(* CoDeSys 2.3.9.41 project: VOS_Vorkuta_ASU_2_osmos_1.pro *)
(* Libraries: PID_Regulators.lib 6.11.19 15:29:27, Util.lib 18.5.10 15:14:28, STANDARD.LIB 4.10.05 11:14:46, IECSFC.LIB 13.4.06 15:51:28, GermesLib_1_4.lib 25.4.21 16:11:00, SYSLIBTIME.LIB 6.11.19 15:29:28, ANALYZATION.LIB 5.10.99 09:05:06 *)

(* PLC configuration (modules and I/O channels)
Fast discrete inputs [I_SIMPLE_INPUT] node 0, in %IB0 out %QB0 {ChannellName = Fast discrete inputs; Filtrationtime = 10000}
  DD1_DI_1 AT %IX0.0 [BitInput] Авария насоса Р03.01/01 {ChannellName = Enter name}
  DD1_DI_2 AT %IX0.1 [BitInput] Авария насоса Р03.01/02 {ChannellName = Enter name}
  DD1_DI_3 AT %IX0.2 [BitInput] эк.манометр PIS03.01/01 после насоса Р03.01/01 {ChannellName = Enter name}
  DD1_DI_4 AT %IX0.3 [BitInput] эк.манометр PIS03.01/02 после насоса Р03.01/02 {ChannellName = Enter name}
Discrete inputs [ID130] node 1, in %IB1 out %QB1 {ChannellName = Discrete inputs; Filtrationtime_GeneralINP = 10; PinCount = 12; Visibility = No}
  AT %IB1.0 [ByteInput] 8 discrete inputs {ChannellName = Enter name}
  AT %IB1.1 [ByteInput] 4 discrete inputs {ChannellName = Enter name}
Fast discrete outputs [OWEN_ID570] node 2, in %IB2 out %QB2 {ChannellName = Fast discrete outputs; SafeValueBool = FALSE; SafeValueBool = FALSE; SafeValueBool = FALSE; SafeValueBool = FALSE; Visibility = No}
  DD1_DO_1 AT %QX2.0 [BitOutput] Fast discrete output 1 {ChannellName = Enter name}
  DD1_DO_2 AT %QX2.1 [BitOutput] Fast discrete output 2 {ChannellName = Enter name}
  DD1_DO_3 AT %QX2.2 [BitOutput] Fast discrete output 3 {ChannellName = Enter name}
  DD1_DO_4 AT %QX2.3 [BitOutput] Fast discrete output 4 {ChannellName = Enter name}
Discrete outputs [ID131] node 3, in %IB3 out %QB3 {ChannellName = Discrete outputs; SafeValueByte = 0; Visibility = No}
  AT %QB3.0 [ByteOutput] 8 discrete outputs {ChannellName = Enter name}
  AT %QB3.1 [ByteOutput] 8 discrete outputs {ChannellName = Enter name}
Fast analog inputs [ID125] node 4, in %IB4 out %QB4 {ChannellName = Fast analog inputs; Flt_Comm = 50Hz 2Por}
  DD1_AI_1 AT %IR4.0 [FloatInputP] LT02.03 уровень в емкости V02.07 {ChannellName = Fast analog input; AIN_TYPE = 0-20 mA; Peak_Filtr = 200; Flt_Ch = Off; TauRC = 10; MinFV = 0; MaxFV = 20}
  DD1_AI_2 AT %IR4.1 [FloatInputP] датчик давления РТ03.01/01 {ChannellName = Fast analog input; AIN_TYPE = 0-20 mA; Peak_Filtr = 200; Flt_Ch = Off; TauRC = 10; MinFV = 0; MaxFV = 20}
  DD1_AI_3 AT %IR4.2 [FloatInputP] датчик давления РТ03.02/01 {ChannellName = Fast analog input; AIN_TYPE = 0-20 mA; Peak_Filtr = 200; Flt_Ch = Off; TauRC = 10; MinFV = 0; MaxFV = 20}
  DD1_AI_4 AT %IR4.3 [FloatInputP] датчик давления РТ03.03/01 {ChannellName = Fast analog input; AIN_TYPE = 0-20 mA; Peak_Filtr = 200; Flt_Ch = Off; TauRC = 10; MinFV = 0; MaxFV = 20}
  DD1_AI_5 AT %IR4.4 [FloatInputP] датчик давления РТ03.04/01 {ChannellName = Fast analog input; AIN_TYPE = 0-20 mA; Peak_Filtr = 200; Flt_Ch = Off; TauRC = 10; MinFV = 0; MaxFV = 20}
  DD1_AI_6 AT %IR4.5 [FloatInputP] кондуктомер QIT03.01/01 осн.осмос {ChannellName = Fast analog input; AIN_TYPE = 0-20 mA; Peak_Filtr = 200; Flt_Ch = Off; TauRC = 10; MinFV = 0; MaxFV = 20}
  DD1_AI_7 AT %IR4.6 [FloatInputP] расходомер FIT03.02/01 осн.осмос {ChannellName = Fast analog input; AIN_TYPE = 0-20 mA; Peak_Filtr = 200; Flt_Ch = Off; TauRC = 10; MinFV = 0; MaxFV = 20}
  DD1_AI_8 AT %IR4.7 [FloatInputP] расходомер FIT03.03/01 осн.осмос {ChannellName = Fast analog input; AIN_TYPE = 0-20 mA; Peak_Filtr = 200; Flt_Ch = Off; TauRC = 10; MinFV = 0; MaxFV = 20}
  AT %IW4.8 [WordInput] AI read time (10ms) {ChannellName = Enter name}
Analog outputs [ID126] node 5, in %IB5 out %QB5 {ChannellName = Analog outputs}
  DD1_AO_1 AT %QR5.0 [FloatOutputP] производительность осн.доз.насоса Р03.02/01 {ChannellName = Analog output; AOUT_TYPE = 4-20 mA; SafeValueREAL = 0.0}
  DD1_AO_2 AT %QR5.1 [FloatOutputP] производительность рез.доз.насоса Р03.02/02 {ChannellName = Analog output; AOUT_TYPE = 4-20 mA; SafeValueREAL = 0.0}
  DD1_AO_3 AT %QR5.2 [FloatOutputP] резерв {ChannellName = Analog output; AOUT_TYPE = 4-20 mA; SafeValueREAL = 0.0}
  DD1_AO_4 AT %QR5.3 [FloatOutputP] резерв {ChannellName = Analog output; AOUT_TYPE = 4-20 mA; SafeValueREAL = 0.0}
Special input [ID103] node 6, in %IB6 out %QB6 {ChannellName = Special input}
  AT %IX6.0 [BitInput] Special input {ChannellName = Enter name}
Special output [ID104] node 7, in %IB7 out %QB7 {ChannellName = Special output}
  AT %QX7.0 [BitOutput] Special output {ChannellName = Enter name}
ModBus (Master) [MODBUS_MASTER_ID450] node 8, in %IB8 out %QB8 {ChannellName = ModBus (Master); Visibility = No}
  AT %QD8.0 [DWordOutput] Last address {ChannellName = Enter name}
  AT %QW8.1 [WordOutput] Last error {ChannellName = Enter name}
  RS-485-1 [COM1_USART] node 0, in %IB8.0 out %QB8.0 {ChannellName = RS-485-1; CommunicationSpeed = 9600; Parity = NO PARITY CHECK; BitLength = 8 bits; StopLength = One stop bit; InterfaceType = RS485; FrameOriented = RTU; Timeout = 5; Visibility = No}
  Universal Modbus device [ID2000] node 1, in %IB8.1 out %QB8.1 {ChannellName = Universal Modbus device; ModuleIP = 10:0:0:223; ServiceTimeout = 150; TCPport = 502; NetMode = Serial; ModuleSlaveAddress = 11; RequestType = By poll time; PeriodOfService = 100; Visibility = No; RepeatCounter = 0; ByteSequence = Native}
    AT %QB8.1.0 [ComChannel] Command (0xff - Start) {ChannellName = Enter name}
    Real input module [ID2007] node 0, in %IB8.1.0 out %QB8.1.0 {ChannellName = float input module; ModbusAddress = 512; Command_read_regs = Read holding Registers  (0x03); Visibility = No}
      PT030102rawValue AT %QD8.1.0.0 [FloatOutput] {ChannellName = Enter name}
    Real input module [ID2007] node 1, in %IB8.1.1 out %QB8.1.1 {ChannellName = float input module; ModbusAddress = 514; Command_read_regs = Read holding Registers  (0x03); Visibility = No}
      PT030202rawValue AT %QD8.1.1.0 [FloatOutput] {ChannellName = Enter name}
    Real input module [ID2007] node 2, in %IB8.1.2 out %QB8.1.2 {ChannellName = float input module; ModbusAddress = 516; Command_read_regs = Read holding Registers  (0x03); Visibility = No}
      PT030302rawValue AT %QD8.1.2.0 [FloatOutput] {ChannellName = Enter name}
    Real input module [ID2007] node 3, in %IB8.1.3 out %QB8.1.3 {ChannellName = float input module; ModbusAddress = 518; Command_read_regs = Read holding Registers  (0x03); Visibility = No}
      PT030402rawValue AT %QD8.1.3.0 [FloatOutput] {ChannellName = Enter name}
    Real input module [ID2007] node 4, in %IB8.1.4 out %QB8.1.4 {ChannellName = float input module; ModbusAddress = 520; Command_read_regs = Read holding Registers  (0x03); Visibility = No}
      QIT030102rawValue AT %QD8.1.4.0 [FloatOutput] {ChannellName = Enter name}
    Real input module [ID2007] node 5, in %IB8.1.5 out %QB8.1.5 {ChannellName = float input module; ModbusAddress = 522; Command_read_regs = Read holding Registers  (0x03); Visibility = No}
      FIT030202rawValue AT %QD8.1.5.0 [FloatOutput] {ChannellName = Enter name}
    Real input module [ID2007] node 6, in %IB8.1.6 out %QB8.1.6 {ChannellName = float input module; ModbusAddress = 524; Command_read_regs = Read holding Registers  (0x03); Visibility = No}
      FIT030302rawValue AT %QD8.1.6.0 [FloatOutput] {ChannellName = Enter name}
      reserve_FIT030101rawValue AT %QD8.1.7.0 [FloatOutput] {ChannellName = Enter name}
    Register input module [ID2003] node 8, in %IB8.1.8 out %QB8.1.8 {ChannellName = Register input module; ModbusAddress = 529; Command_read_regs = Read input registers  (0x04); Visibility = No}
      DI_bit_mask_DD2 AT %QW8.1.8.0 [WordOutput] {ChannellName = Enter name}
    Register input module [ID2003] node 9, in %IB8.1.9 out %QB8.1.9 {ChannellName = Register input module; ModbusAddress = 532; Command_read_regs = Read input registers  (0x04); Visibility = No}
      stat_word_P030601_PLC AT %QW8.1.9.0 [WordOutput] {ChannellName = Enter name}
    Register input module [ID2003] node 10, in %IB8.1.10 out %QB8.1.10 {ChannellName = Register input module; ModbusAddress = 535; Command_read_regs = Read input registers  (0x04); Visibility = No}
      stat_word_P030602_PLC AT %QW8.1.10.0 [WordOutput] {ChannellName = Enter name}
  Universal Modbus device [ID2000] node 2, in %IB8.2 out %QB8.2 {ChannellName = Universal Modbus device; ModuleIP = 10:0:0:223; ServiceTimeout = 150; TCPport = 502; NetMode = Serial; ModuleSlaveAddress = 1; RequestType = By value change; PeriodOfService = 100; Visibility = No; RepeatCounter = 0; ByteSequence = Native}
    AT %QB8.2.0 [ComChannel] Command (0xff - Start) {ChannellName = Enter name}
    Register output module [ID2004] node 0, in %IB8.2.0 out %QB8.2.0 {ChannellName = Register; ModbusAddress = 528; Command_write_one_reg = Write multiple registers(0x10); Visibility = No}
      DO_bit_mask_DD2 AT %QW8.2.0.0 [WordOutput] {ChannellName = Enter name}
    Register output module [ID2004] node 1, in %IB8.2.1 out %QB8.2.1 {ChannellName = Register; ModbusAddress = 530; Command_write_one_reg = Write multiple registers(0x10); Visibility = No}
      com_word_P030601_PLC AT %QW8.2.1.0 [WordOutput] {ChannellName = Enter name}
    Register output module [ID2004] node 2, in %IB8.2.2 out %QB8.2.2 {ChannellName = Register; ModbusAddress = 531; Command_write_one_reg = Write multiple registers(0x10); Visibility = No}
      set_freq_P030601_PLC AT %QW8.2.2.0 [WordOutput] {ChannellName = Enter name}
    Register output module [ID2004] node 3, in %IB8.2.3 out %QB8.2.3 {ChannellName = Register; ModbusAddress = 533; Command_write_one_reg = Write multiple registers(0x10); Visibility = No}
      com_word_P030602_PLC AT %QW8.2.3.0 [WordOutput] {ChannellName = Enter name}
    Register output module [ID2004] node 4, in %IB8.2.4 out %QB8.2.4 {ChannellName = Register; ModbusAddress = 534; Command_write_one_reg = Write multiple registers(0x10); Visibility = No}
      set_freq_P030602_PLC AT %QW8.2.4.0 [WordOutput] {ChannellName = Enter name}
ModBus (Master) [MODBUS_MASTER_ID450] node 9, in %IB9 out %QB9 {ChannellName = ModBus (Master); Visibility = No}
  AT %QD9.0 [DWordOutput] Last address {ChannellName = Enter name}
  AT %QW9.1 [WordOutput] Last error {ChannellName = Enter name}
  RS-232 [COM2_USART] node 0, in %IB9.0 out %QB9.0 {ChannellName = RS-232; CommunicationSpeed = 115200; Parity = NO PARITY CHECK; BitLength = 8 bits; StopLength = One stop bit; InterfaceType = RS232; FrameOriented = RTU; Timeout = 5; Visibility = No}
  Universal Modbus device [ID2000] node 1, in %IB9.1 out %QB9.1 {ChannellName = Universal Modbus device; ModuleIP = 10:0:0:223; ServiceTimeout = 150; TCPport = 502; NetMode = Serial; ModuleSlaveAddress = 1; RequestType = By poll time; PeriodOfService = 50; Visibility = No; RepeatCounter = 0; ByteSequence = Native}
    AT %QB9.1.0 [ComChannel] Command (0xff - Start) {ChannellName = Enter name}
PANsetWordP0302 AT %QW9.1.0.0 [WordOutput] {ChannellName = Enter name}
PAN_LT0203maxValue AT %QD9.1.1.0 [FloatOutput] {ChannellName = Enter name}
PANsetMaxPumpDosingValueP0302 AT %QD9.1.2.0 [FloatOutput] {ChannellName = Enter name}
PANsetKoeffPropotrionalityP0302 AT %QD9.1.3.0 [FloatOutput] {ChannellName = Enter name}
PAN_CHECKING_DELAY_TIME AT %QW9.1.4.0 [WordOutput] {ChannellName = Enter name}
PAN_DELAY_REPEATED_START_SEC AT %QW9.1.5.0 [WordOutput] {ChannellName = Enter name}
PAN_DELAY_TO_OFF_VALVE AT %QW9.1.6.0 [WordOutput] {ChannellName = Enter name}
PAN_DELAY_TO_CHECK_PT0301 AT %QW9.1.7.0 [WordOutput] {ChannellName = Enter name}
PAN_DELAY_TO_SWITCH_VALVE AT %QW9.1.8.0 [WordOutput] {ChannellName = Enter name}
PAN_DELAY_TO_CLOSE_VALVE AT %QW9.1.9.0 [WordOutput] {ChannellName = Enter name}
PAN_FIT030201maxValue AT %QD9.1.10.0 [FloatOutput] {ChannellName = Enter name}
PAN_FIT030301maxValue AT %QD9.1.11.0 [FloatOutput] {ChannellName = Enter name}
PAN_FIT030202maxValue AT %QD9.1.12.0 [FloatOutput] {ChannellName = Enter name}
PAN_FIT030302maxValue AT %QD9.1.13.0 [FloatOutput] {ChannellName = Enter name}
PAN_QIT030101maxValue AT %QD9.1.14.0 [FloatOutput] {ChannellName = Enter name}
PAN_QIT030102maxValue AT %QD9.1.15.0 [FloatOutput] {ChannellName = Enter name}
PAN_PT030101maxValue AT %QD9.1.16.0 [FloatOutput] {ChannellName = Enter name}
PAN_PT030201maxValue AT %QD9.1.17.0 [FloatOutput] {ChannellName = Enter name}
PAN_PT030301maxValue AT %QD9.1.18.0 [FloatOutput] {ChannellName = Enter name}
PAN_PT030401maxValue AT %QD9.1.19.0 [FloatOutput] {ChannellName = Enter name}
PAN_PT030102maxValue AT %QD9.1.20.0 [FloatOutput] {ChannellName = Enter name}
PAN_PT030202maxValue AT %QD9.1.21.0 [FloatOutput] {ChannellName = Enter name}
PAN_PT030302maxValue AT %QD9.1.22.0 [FloatOutput] {ChannellName = Enter name}
PAN_PT030402maxValue AT %QD9.1.23.0 [FloatOutput] {ChannellName = Enter name}
PANsetWordOsmos AT %QW9.1.24.0 [WordOutput] {ChannellName = Enter name}
PAN_PT0301startValue AT %QD9.1.25.0 [FloatOutput] {ChannellName = Enter name}
PAN_FIT0303setValue AT %QD9.1.26.0 [FloatOutput] {ChannellName = Enter name}
PAN_PT0302setMaxValue AT %QD9.1.27.0 [FloatOutput] {ChannellName = Enter name}
PAN_PT0303setMaxValue AT %QD9.1.28.0 [FloatOutput] {ChannellName = Enter name}
PAN_PT0304setMaxValue AT %QD9.1.29.0 [FloatOutput] {ChannellName = Enter name}
PAN_KP_F_P030601 AT %QD9.1.30.0 [FloatOutput] {ChannellName = Enter name}
PAN_I_F_P030601 AT %QD9.1.31.0 [FloatOutput] {ChannellName = Enter name}
%MPAN_D_F_P030601 AT %QD9.1.32.0 [FloatOutput] {ChannellName = Enter name}
%MPAN_KP_P_P030601 AT %QD9.1.33.0 [FloatOutput] {ChannellName = Enter name}
PAN_I_P_P030601 AT %QD9.1.34.0 [FloatOutput] {ChannellName = Enter name}
PAN_D_P_P030601 AT %QD9.1.35.0 [FloatOutput] {ChannellName = Enter name}
PAN_KP_F_P030602 AT %QD9.1.36.0 [FloatOutput] {ChannellName = Enter name}
PAN_I_F_P030602 AT %QD9.1.37.0 [FloatOutput] {ChannellName = Enter name}
PAN_D_F_P030602 AT %QD9.1.38.0 [FloatOutput] {ChannellName = Enter name}
PAN_KP_P_P030602 AT %QD9.1.39.0 [FloatOutput] {ChannellName = Enter name}
PAN_I_P_P030602 AT %QD9.1.40.0 [FloatOutput] {ChannellName = Enter name}
PAN_D_P_P030602 AT %QD9.1.41.0 [FloatOutput] {ChannellName = Enter name}
PAN_FIT0303_SetCascade AT %QD9.1.42.0 [FloatOutput] {ChannellName = Enter name}
ID2003NoNoINTRegister input module+ AT %QW9.1.43.0 [WordOutput] B	+%QB	+%MB	+%MPAN_valuesActivator {ChannellName = Enter name}
PAN_V0207maxHeight AT %QD9.1.44.0 [FloatOutput] {ChannellName = Enter name}
PAN_V0207minHeight AT %QD9.1.45.0 [FloatOutput] {ChannellName = Enter name}
Universal Modbus device [ID2000] node 2, in %IB9.2 out %QB9.2 {ChannellName = Universal Modbus device; ModuleIP = 10:0:0:223; ServiceTimeout = 150; TCPport = 502; NetMode = Serial; ModuleSlaveAddress = 1; RequestType = Both; PeriodOfService = 100; Visibility = No; RepeatCounter = 0; ByteSequence = Native}
  AT %QB9.2.0 [ComChannel] Command (0xff - Start) {ChannellName = Enter name}
  Register output module [ID2004] node 0, in %IB9.2.0 out %QB9.2.0 {ChannellName = Register; ModbusAddress = 271; Command_write_one_reg = Write multiple registers(0x10); Visibility = No}
    PANstatWordP0302 AT %QW9.2.0.0 [WordOutput] {ChannellName = Enter name}
  Register output module [ID2004] node 1, in %IB9.2.1 out %QB9.2.1 {ChannellName = Register; ModbusAddress = 272; Command_write_one_reg = Write multiple registers(0x10); Visibility = No}
    PANdaysOfWorkP030201 AT %QW9.2.1.0 [WordOutput] {ChannellName = Enter name}
  Register output module [ID2004] node 2, in %IB9.2.2 out %QB9.2.2 {ChannellName = Register; ModbusAddress = 273; Command_write_one_reg = Write multiple registers(0x10); Visibility = No}
    PANhoursOfWorkP030201 AT %QW9.2.2.0 [WordOutput] {ChannellName = Enter name}
  Register output module [ID2004] node 3, in %IB9.2.3 out %QB9.2.3 {ChannellName = Register; ModbusAddress = 274; Command_write_one_reg = Write multiple registers(0x10); Visibility = No}
    PANminutesOfWorkP030201 AT %QW9.2.3.0 [WordOutput] {ChannellName = Enter name}
  Register output module [ID2004] node 4, in %IB9.2.4 out %QB9.2.4 {ChannellName = Register; ModbusAddress = 275; Command_write_one_reg = Write multiple registers(0x10); Visibility = No}
    PANsecondsOfWorkP030201 AT %QW9.2.4.0 [WordOutput] {ChannellName = Enter name}
  Register output module [ID2004] node 5, in %IB9.2.5 out %QB9.2.5 {ChannellName = Register; ModbusAddress = 276; Command_write_one_reg = Write multiple registers(0x10); Visibility = No}
    PANtoNextStartP030201timer AT %QW9.2.5.0 [WordOutput] {ChannellName = Enter name}
  Register output module [ID2004] node 6, in %IB9.2.6 out %QB9.2.6 {ChannellName = Register; ModbusAddress = 277; Command_write_one_reg = Write multiple registers(0x10); Visibility = No}
    PANdaysOfWorkP030202 AT %QW9.2.6.0 [WordOutput] {ChannellName = Enter name}
  Register output module [ID2004] node 7, in %IB9.2.7 out %QB9.2.7 {ChannellName = Register; ModbusAddress = 278; Command_write_one_reg = Write multiple registers(0x10); Visibility = No}
    PANhoursOfWorkP030202 AT %QW9.2.7.0 [WordOutput] {ChannellName = Enter name}
  Register output module [ID2004] node 8, in %IB9.2.8 out %QB9.2.8 {ChannellName = Register; ModbusAddress = 279; Command_write_one_reg = Write multiple registers(0x10); Visibility = No}
    PANminutesOfWorkP030202 AT %QW9.2.8.0 [WordOutput] {ChannellName = Enter name}
  Register output module [ID2004] node 9, in %IB9.2.9 out %QB9.2.9 {ChannellName = Register; ModbusAddress = 280; Command_write_one_reg = Write multiple registers(0x10); Visibility = No}
    PANsecondsOfWorkP030202 AT %QW9.2.9.0 [WordOutput] {ChannellName = Enter name}
  Register output module [ID2004] node 10, in %IB9.2.10 out %QB9.2.10 {ChannellName = Register; ModbusAddress = 281; Command_write_one_reg = Write multiple registers(0x10); Visibility = No}
    PANtoNextStartP030202timer AT %QW9.2.10.0 [WordOutput] {ChannellName = Enter name}
  Real output module [ID2008] node 11, in %IB9.2.11 out %QB9.2.11 {ChannellName = float output module; ModbusAddress = 282; Command_write_regs = Preset multiple Registers (0x10); Visibility = No}
    PANcounterP030201 AT %QD9.2.11.0 [FloatOutput] {ChannellName = Enter name}
  Real output module [ID2008] node 12, in %IB9.2.12 out %QB9.2.12 {ChannellName = float output module; ModbusAddress = 284; Command_write_regs = Preset multiple Registers (0x10); Visibility = No}
    PANcounterP030202 AT %QD9.2.12.0 [FloatOutput] {ChannellName = Enter name}
  Real output module [ID2008] node 13, in %IB9.2.13 out %QB9.2.13 {ChannellName = float output module; ModbusAddress = 286; Command_write_regs = Preset multiple Registers (0x10); Visibility = No}
    PAN_FIT0301realValue AT %QD9.2.13.0 [FloatOutput] {ChannellName = Enter name}
  Real output module [ID2008] node 14, in %IB9.2.14 out %QB9.2.14 {ChannellName = float output module; ModbusAddress = 288; Command_write_regs = Preset multiple Registers (0x10); Visibility = No}
    PAN_PT030101realValue AT %QD9.2.14.0 [FloatOutput] {ChannellName = Enter name}
  Real output module [ID2008] node 15, in %IB9.2.15 out %QB9.2.15 {ChannellName = float output module; ModbusAddress = 290; Command_write_regs = Preset multiple Registers (0x10); Visibility = No}
    PAN_PT030201realValue AT %QD9.2.15.0 [FloatOutput] {ChannellName = Enter name}
  Real output module [ID2008] node 16, in %IB9.2.16 out %QB9.2.16 {ChannellName = float output module; ModbusAddress = 292; Command_write_regs = Preset multiple Registers (0x10); Visibility = No}
    PAN_PT030301realValue AT %QD9.2.16.0 [FloatOutput] {ChannellName = Enter name}
  Real output module [ID2008] node 17, in %IB9.2.17 out %QB9.2.17 {ChannellName = float output module; ModbusAddress = 294; Command_write_regs = Preset multiple Registers (0x10); Visibility = No}
    PAN_FIT030301realValue AT %QD9.2.17.0 [FloatOutput] {ChannellName = Enter name}
  Real output module [ID2008] node 18, in %IB9.2.18 out %QB9.2.18 {ChannellName = float output module; ModbusAddress = 296; Command_write_regs = Preset multiple Registers (0x10); Visibility = No}
    PAN_PT030102realValue AT %QD9.2.18.0 [FloatOutput] {ChannellName = Enter name}
  Real output module [ID2008] node 19, in %IB9.2.19 out %QB9.2.19 {ChannellName = float output module; ModbusAddress = 298; Command_write_regs = Preset multiple Registers (0x10); Visibility = No}
    PAN_PT030202realValue AT %QD9.2.19.0 [FloatOutput] {ChannellName = Enter name}
  Real output module [ID2008] node 20, in %IB9.2.20 out %QB9.2.20 {ChannellName = float output module; ModbusAddress = 300; Command_write_regs = Preset multiple Registers (0x10); Visibility = No}
    PAN_PT030302realValue AT %QD9.2.20.0 [FloatOutput] {ChannellName = Enter name}
  Real output module [ID2008] node 21, in %IB9.2.21 out %QB9.2.21 {ChannellName = float output module; ModbusAddress = 302; Command_write_regs = Preset multiple Registers (0x10); Visibility = No}
    PAN_FIT030302realValue AT %QD9.2.21.0 [FloatOutput] {ChannellName = Enter name}
  Real output module [ID2008] node 22, in %IB9.2.22 out %QB9.2.22 {ChannellName = float output module; ModbusAddress = 304; Command_write_regs = Preset multiple Registers (0x10); Visibility = No}
    PAN_PT030401realValue AT %QD9.2.22.0 [FloatOutput] {ChannellName = Enter name}
  Real output module [ID2008] node 23, in %IB9.2.23 out %QB9.2.23 {ChannellName = float output module; ModbusAddress = 306; Command_write_regs = Preset multiple Registers (0x10); Visibility = No}
    PAN_FIT030201realValue AT %QD9.2.23.0 [FloatOutput] {ChannellName = Enter name}
  Real output module [ID2008] node 24, in %IB9.2.24 out %QB9.2.24 {ChannellName = float output module; ModbusAddress = 308; Command_write_regs = Preset multiple Registers (0x10); Visibility = No}
    PAN_QIT030101realValue AT %QD9.2.24.0 [FloatOutput] {ChannellName = Enter name}
  Real output module [ID2008] node 25, in %IB9.2.25 out %QB9.2.25 {ChannellName = float output module; ModbusAddress = 310; Command_write_regs = Preset multiple Registers (0x10); Visibility = No}
    PAN_PT030402realValue AT %QD9.2.25.0 [FloatOutput] {ChannellName = Enter name}
  Real output module [ID2008] node 26, in %IB9.2.26 out %QB9.2.26 {ChannellName = float output module; ModbusAddress = 312; Command_write_regs = Preset multiple Registers (0x10); Visibility = No}
    PAN_FIT030202realValue AT %QD9.2.26.0 [FloatOutput] {ChannellName = Enter name}
  Real output module [ID2008] node 27, in %IB9.2.27 out %QB9.2.27 {ChannellName = float output module; ModbusAddress = 314; Command_write_regs = Preset multiple Registers (0x10); Visibility = No}
    PAN_QIT030102realValue AT %QD9.2.27.0 [FloatOutput] {ChannellName = Enter name}
  Register output module [ID2004] node 28, in %IB9.2.28 out %QB9.2.28 {ChannellName = Register; ModbusAddress = 316; Command_write_one_reg = Write multiple registers(0x10); Visibility = No}
    PANstatWordOsmos AT %QW9.2.28.0 [WordOutput] {ChannellName = Enter name}
  Register output module [ID2004] node 29, in %IB9.2.29 out %QB9.2.29 {ChannellName = Register; ModbusAddress = 317; Command_write_one_reg = Write multiple registers(0x10); Visibility = No}
    PANdaysOfWorkOsmos1 AT %QW9.2.29.0 [WordOutput] {ChannellName = Enter name}
  Register output module [ID2004] node 30, in %IB9.2.30 out %QB9.2.30 {ChannellName = Register; ModbusAddress = 318; Command_write_one_reg = Write multiple registers(0x10); Visibility = No}
    PANhoursOfWorkOsmos1 AT %QW9.2.30.0 [WordOutput] {ChannellName = Enter name}
  Register output module [ID2004] node 31, in %IB9.2.31 out %QB9.2.31 {ChannellName = Register; ModbusAddress = 319; Command_write_one_reg = Write multiple registers(0x10); Visibility = No}
    PANminutesOfWorkOsmos1 AT %QW9.2.31.0 [WordOutput] {ChannellName = Enter name}
  Register output module [ID2004] node 32, in %IB9.2.32 out %QB9.2.32 {ChannellName = Register; ModbusAddress = 320; Command_write_one_reg = Write multiple registers(0x10); Visibility = No}
    PANsecondsOfWorkOsmos1 AT %QW9.2.32.0 [WordOutput] {ChannellName = Enter name}
  Register output module [ID2004] node 33, in %IB9.2.33 out %QB9.2.33 {ChannellName = Register; ModbusAddress = 321; Command_write_one_reg = Write multiple registers(0x10); Visibility = No}
    PANtoNextStartOsmos1timer AT %QW9.2.33.0 [WordOutput] {ChannellName = Enter name}
  Real output module [ID2008] node 34, in %IB9.2.34 out %QB9.2.34 {ChannellName = float output module; ModbusAddress = 322; Command_write_regs = Preset multiple Registers (0x10); Visibility = No}
    PANcounterOsmos1 AT %QD9.2.34.0 [FloatOutput] {ChannellName = Enter name}
  Real output module [ID2008] node 35, in %IB9.2.35 out %QB9.2.35 {ChannellName = float output module; ModbusAddress = 324; Command_write_regs = Preset multiple Registers (0x10); Visibility = No}
    PANcounterOsmos2 AT %QD9.2.35.0 [FloatOutput] {ChannellName = Enter name}
  Register output module [ID2004] node 36, in %IB9.2.36 out %QB9.2.36 {ChannellName = Register; ModbusAddress = 326; Command_write_one_reg = Write multiple registers(0x10); Visibility = No}
    PANdaysOfWorkOsmos2 AT %QW9.2.36.0 [WordOutput] {ChannellName = Enter name}
  Register output module [ID2004] node 37, in %IB9.2.37 out %QB9.2.37 {ChannellName = Register; ModbusAddress = 327; Command_write_one_reg = Write multiple registers(0x10); Visibility = No}
    PANhoursOfWorkOsmos2 AT %QW9.2.37.0 [WordOutput] {ChannellName = Enter name}
  Register output module [ID2004] node 38, in %IB9.2.38 out %QB9.2.38 {ChannellName = Register; ModbusAddress = 328; Command_write_one_reg = Write multiple registers(0x10); Visibility = No}
    PANminutesOfWorkOsmos2 AT %QW9.2.38.0 [WordOutput] {ChannellName = Enter name}
  Register output module [ID2004] node 39, in %IB9.2.39 out %QB9.2.39 {ChannellName = Register; ModbusAddress = 329; Command_write_one_reg = Write multiple registers(0x10); Visibility = No}
    PANsecondsOfWorkOsmos2 AT %QW9.2.39.0 [WordOutput] {ChannellName = Enter name}
  Register output module [ID2004] node 40, in %IB9.2.40 out %QB9.2.40 {ChannellName = Register; ModbusAddress = 330; Command_write_one_reg = Write multiple registers(0x10); Visibility = No}
    PANtoNextStartOsmos2timer AT %QW9.2.40.0 [WordOutput] {ChannellName = Enter name}
  Register output module [ID2004] node 41, in %IB9.2.41 out %QB9.2.41 {ChannellName = Register; ModbusAddress = 331; Command_write_one_reg = Write multiple registers(0x10); Visibility = No}
    PANmainViewBools AT %QW9.2.41.0 [WordOutput] {ChannellName = Enter name}
PAN_BMT_Flow AT %QD9.2.42.0 [FloatOutput] {ChannellName = Enter name}
32bit output module [ID2006] node 43, in %IB9.2.43 out %QB9.2.43 {ChannellName = 32 bit output module; ModbusAddress = 336; Command_write_regs = Preset multiple Registers (0x10); Visibility = No}
  PANalarms AT %QD9.2.43.0 [DWordOutput] {ChannellName = Enter name}
Real output module [ID2008] node 44, in %IB9.2.44 out %QB9.2.44 {ChannellName = float output module; ModbusAddress = 338; Command_write_regs = Preset multiple Registers (0x10); Visibility = No}
  PAN_currentValue_PT0301startValue AT %QD9.2.44.0 [FloatOutput] {ChannellName = Enter name}
Real output module [ID2008] node 45, in %IB9.2.45 out %QB9.2.45 {ChannellName = float output module; ModbusAddress = 340; Command_write_regs = Preset multiple Registers (0x10); Visibility = No}
  PAN_currentValue_FIT0303setValue AT %QD9.2.45.0 [FloatOutput] {ChannellName = Enter name}
Real output module [ID2008] node 46, in %IB9.2.46 out %QB9.2.46 {ChannellName = float output module; ModbusAddress = 342; Command_write_regs = Preset multiple Registers (0x10); Visibility = No}
  PAN_currentValue_PT0302setMaxValue AT %QD9.2.46.0 [FloatOutput] {ChannellName = Enter name}
Real output module [ID2008] node 47, in %IB9.2.47 out %QB9.2.47 {ChannellName = float output module; ModbusAddress = 344; Command_write_regs = Preset multiple Registers (0x10); Visibility = No}
  PAN_currentValue_PT0303setMaxValue AT %QD9.2.47.0 [FloatOutput] {ChannellName = Enter name}
Real output module [ID2008] node 48, in %IB9.2.48 out %QB9.2.48 {ChannellName = float output module; ModbusAddress = 346; Command_write_regs = Preset multiple Registers (0x10); Visibility = No}
  PAN_currentValue_PT0304setMaxValue AT %QD9.2.48.0 [FloatOutput] {ChannellName = Enter name}
Real output module [ID2008] node 49, in %IB9.2.49 out %QB9.2.49 {ChannellName = float output module; ModbusAddress = 348; Command_write_regs = Preset multiple Registers (0x10); Visibility = No}
  PAN_currentValue_FIT0303_SetCascade AT %QD9.2.49.0 [FloatOutput] {ChannellName = Enter name}
Real output module [ID2008] node 50, in %IB9.2.50 out %QB9.2.50 {ChannellName = float output module; ModbusAddress = 350; Command_write_regs = Preset multiple Registers (0x10); Visibility = No}
  PAN_currentValue_KP_F_P030601 AT %QD9.2.50.0 [FloatOutput] {ChannellName = Enter name}
Real output module [ID2008] node 51, in %IB9.2.51 out %QB9.2.51 {ChannellName = float output module; ModbusAddress = 352; Command_write_regs = Preset multiple Registers (0x10); Visibility = No}
  PAN_currentValue_I_F_P030601 AT %QD9.2.51.0 [FloatOutput] {ChannellName = Enter name}
Real output module [ID2008] node 52, in %IB9.2.52 out %QB9.2.52 {ChannellName = float output module; ModbusAddress = 354; Command_write_regs = Preset multiple Registers (0x10); Visibility = No}
  PAN_currentValue_D_F_P030601 AT %QD9.2.52.0 [FloatOutput] {ChannellName = Enter name}
Real output module [ID2008] node 53, in %IB9.2.53 out %QB9.2.53 {ChannellName = float output module; ModbusAddress = 356; Command_write_regs = Preset multiple Registers (0x10); Visibility = No}
  PAN_currentValue_KP_P_P030601 AT %QD9.2.53.0 [FloatOutput] {ChannellName = Enter name}
Real output module [ID2008] node 54, in %IB9.2.54 out %QB9.2.54 {ChannellName = float output module; ModbusAddress = 358; Command_write_regs = Preset multiple Registers (0x10); Visibility = No}
  PAN_currentValue_I_P_P030601 AT %QD9.2.54.0 [FloatOutput] {ChannellName = Enter name}
Real output module [ID2008] node 55, in %IB9.2.55 out %QB9.2.55 {ChannellName = float output module; ModbusAddress = 360; Command_write_regs = Preset multiple Registers (0x10); Visibility = No}
  PAN_currentValue_D_P_P030601 AT %QD9.2.55.0 [FloatOutput] {ChannellName = Enter name}
Real output module [ID2008] node 56, in %IB9.2.56 out %QB9.2.56 {ChannellName = float output module; ModbusAddress = 362; Command_write_regs = Preset multiple Registers (0x10); Visibility = No}
  PAN_currentValue_KP_F_P030602 AT %QD9.2.56.0 [FloatOutput] {ChannellName = Enter name}
Real output module [ID2008] node 57, in %IB9.2.57 out %QB9.2.57 {ChannellName = float output module; ModbusAddress = 364; Command_write_regs = Preset multiple Registers (0x10); Visibility = No}
  PAN_currentValue_I_F_P030602 AT %QD9.2.57.0 [FloatOutput] {ChannellName = Enter name}
Real output module [ID2008] node 58, in %IB9.2.58 out %QB9.2.58 {ChannellName = float output module; ModbusAddress = 366; Command_write_regs = Preset multiple Registers (0x10); Visibility = No}
  PAN_currentValue_D_F_P030602 AT %QD9.2.58.0 [FloatOutput] {ChannellName = Enter name}
Real output module [ID2008] node 59, in %IB9.2.59 out %QB9.2.59 {ChannellName = float output module; ModbusAddress = 368; Command_write_regs = Preset multiple Registers (0x10); Visibility = No}
  PAN_currentValue_KP_P_P030602 AT %QD9.2.59.0 [FloatOutput] {ChannellName = Enter name}
Real output module [ID2008] node 60, in %IB9.2.60 out %QB9.2.60 {ChannellName = float output module; ModbusAddress = 370; Command_write_regs = Preset multiple Registers (0x10); Visibility = No}
  PAN_currentValue_I_P_P030602 AT %QD9.2.60.0 [FloatOutput] {ChannellName = Enter name}
Real output module [ID2008] node 61, in %IB9.2.61 out %QB9.2.61 {ChannellName = float output module; ModbusAddress = 372; Command_write_regs = Preset multiple Registers (0x10); Visibility = No}
  PAN_currentValue_D_P_P030602 AT %QD9.2.61.0 [FloatOutput] {ChannellName = Enter name}
Real output module [ID2008] node 62, in %IB9.2.62 out %QB9.2.62 {ChannellName = float output module; ModbusAddress = 374; Command_write_regs = Preset multiple Registers (0x10); Visibility = No}
  PAN_currentValue_setMaxPumpDosingValueP0302 AT %QD9.2.62.0 [FloatOutput] {ChannellName = Enter name}
Real output module [ID2008] node 63, in %IB9.2.63 out %QB9.2.63 {ChannellName = float output module; ModbusAddress = 376; Command_write_regs = Preset multiple Registers (0x10); Visibility = No}
  PAN_currentValue_setKoeffProportionalityP0302 AT %QD9.2.63.0 [FloatOutput] {ChannellName = Enter name}
Register output module [ID2004] node 64, in %IB9.2.64 out %QB9.2.64 {ChannellName = Register; ModbusAddress = 378; Command_write_one_reg = Write multiple registers(0x10); Visibility = No}
  PAN_currentValue_CHECKING_DELAY_TIME AT %QW9.2.64.0 [WordOutput] {ChannellName = Enter name}
Register output module [ID2004] node 65, in %IB9.2.65 out %QB9.2.65 {ChannellName = Register; ModbusAddress = 379; Command_write_one_reg = Write multiple registers(0x10); Visibility = No}
  PAN_currentValue_DELAY_REPEATED_START_SEC AT %QW9.2.65.0 [WordOutput] {ChannellName = Enter name}
Register output module [ID2004] node 66, in %IB9.2.66 out %QB9.2.66 {ChannellName = Register; ModbusAddress = 380; Command_write_one_reg = Write multiple registers(0x10); Visibility = No}
  PAN_currentValue_DELAY_TO_OFF_VALVE AT %QW9.2.66.0 [WordOutput] {ChannellName = Enter name}
Register output module [ID2004] node 67, in %IB9.2.67 out %QB9.2.67 {ChannellName = Register; ModbusAddress = 381; Command_write_one_reg = Write multiple registers(0x10); Visibility = No}
  PAN_currentValue_DELAY_TO_CHECK_PT0301 AT %QW9.2.67.0 [WordOutput] {ChannellName = Enter name}
Register output module [ID2004] node 68, in %IB9.2.68 out %QB9.2.68 {ChannellName = Register; ModbusAddress = 382; Command_write_one_reg = Write multiple registers(0x10); Visibility = No}
  PAN_currentValue_DELAY_TO_SWITCH_VALVE AT %QW9.2.68.0 [WordOutput] {ChannellName = Enter name}
Register output module [ID2004] node 69, in %IB9.2.69 out %QB9.2.69 {ChannellName = Register; ModbusAddress = 383; Command_write_one_reg = Write multiple registers(0x10); Visibility = No}
  PAN_currentValue_DELAY_TO_CLOSE_VALVE AT %QW9.2.69.0 [WordOutput] {ChannellName = Enter name}
PAN_currentValue_FIT0301maxValue AT %QD9.2.70.0 [FloatOutput] {ChannellName = Enter name}
PAN_currentValue_FIT030201maxValue AT %QD9.2.71.0 [FloatOutput] {ChannellName = Enter name}
PAN_currentValue_FIT030301maxValue AT %QD9.2.72.0 [FloatOutput] {ChannellName = Enter name}
PAN_currentValue_FIT030202maxValue AT %QD9.2.73.0 [FloatOutput] {ChannellName = Enter name}
PAN_currentValue_FIT030302maxValue AT %QD9.2.74.0 [FloatOutput] {ChannellName = Enter name}
PAN_currentValue_QIT030101maxValue AT %QD9.2.75.0 [FloatOutput] {ChannellName = Enter name}
PAN_currentValue_QIT030102maxValue AT %QD9.2.76.0 [FloatOutput] {ChannellName = Enter name}
PAN_currentValue_PT030101maxValue AT %QD9.2.77.0 [FloatOutput] {ChannellName = Enter name}
PAN_currentValue_PT030201maxValue AT %QD9.2.78.0 [FloatOutput] {ChannellName = Enter name}
PAN_currentValue_PT030301maxValue AT %QD9.2.79.0 [FloatOutput] {ChannellName = Enter name}
PAN_currentValue_PT030401maxValue AT %QD9.2.80.0 [FloatOutput] {ChannellName = Enter name}
PAN_currentValue_PT030102maxValue AT %QD9.2.81.0 [FloatOutput] {ChannellName = Enter name}
PAN_currentValue_PT030202maxValue AT %QD9.2.82.0 [FloatOutput] {ChannellName = Enter name}
PAN_currentValue_PT030302maxValue AT %QD9.2.83.0 [FloatOutput] {ChannellName = Enter name}
PAN_currentValue_PT030402maxValue AT %QD9.2.84.0 [FloatOutput] {ChannellName = Enter name}
PAN_currentValue_LT0203maxValue AT %QD9.2.85.0 [FloatOutput] {ChannellName = Enter name}
PAN_currentValue_V0207minHeight AT %QD9.2.86.0 [FloatOutput] {ChannellName = Enter name}
PAN_currentValue_V0207maxHeight AT %QD9.2.87.0 [FloatOutput] {ChannellName = Enter name}
PAN_currentValue_V0207height AT %QD9.2.88.0 [FloatOutput] {ChannellName = Enter name}
TCP [TCP_ID221] node 0, in %IB10.0.0 out %QB10.0.0 {ChannellName = TCP; RemotePort = 502; Visibility = No}
ASU_FlowFromBMT AT %QD10.1.0 [FloatOutput] {ChannellName = Enter name}
ASU_FlowFIT0102 AT %QD10.2.0 [FloatOutput] {ChannellName = Enter name}
ASU_Levels_input AT %QW10.3.0 [WordOutput] {ChannellName = Enter name}
ASU_Levels_output AT %QW10.4.0 [WordOutput] {ChannellName = Enter name}
*)

(* POU PLC_PRG, CFC *)
PROGRAM PLC_PRG
VAR
	resetAlarms: BOOL;		(*Сброс аварий в осмос 2 (МЕ03)*)
	lowLevelV0207: BOOL;		(*низкий уровень в емкости V02.07, сигнал из АСУ-2 осмос-1*)
	highLevelV0601: BOOL;		(*высокий уровень в емкости V06.01 сигнал из АСУ-1 общий.*)
	FIT0301realValue: REAL;		(*Показания расходомера FIT03.01/01 на входе в осмос 2.
			Для управления производительностью НД Р03.02 (1 и 2).*)
	P0302: RichTwoPumpManager;		(*блок управления доз.насосами Р03.02/01 и Р03.02/02.*)
	P0302dos: DosingPumpProportional;		(*блок управления промзводительностью доз.насосов Р03.02.*)
	dosingErrorP0302: BOOL;		(*Ошибка производительности дозирования (неверно заданы значения производительности насоса,
производительность доз.насоса не соответствует расходу.*)
	initializer: R_TRIG;		(*триггер дающий импульс при включении программы.*)
	alarmP0302: BOOL;		(*авария обоих доз.насосов Р03..02 на входе в осмос*)
	osmosTotalAlarm: BOOL;		(*авария обоих осмосов*)
	controlAIpt030101: ControlAI;
	PT030101realValue: REAL;		(*Показания датчика РТ03.01/01, МПа (Бар)*)
	PT030101alarm: BOOL;		(*авария датчика РТ03.01/01*)
	controlAIpt030201: ControlAI;
	PT030201realValue: REAL;
	PT030201alarm: BOOL;
	controlAIpt030301: ControlAI;
	PT030301realValue: REAL;
	PT030301alarm: BOOL;
	controlAIpt030401: ControlAI;
	PT030401realValue: REAL;
	PT030401alarm: BOOL;
	controlAIqit030101: ControlAI;
	QIT030101realValue: REAL;
	QIT030101alarm: BOOL;
	controlAIfit030201: ControlAI;
	FIT030201realValue: REAL;
	FIT030201alarm: BOOL;
	controlAIfit030301: ControlAI;
	FIT030301realValue: REAL;
	FIT030301alarm: BOOL;
	osmos2sensorsAlarm: BOOL;		(*Авария датчиков осмос 2.
			в DD2 (ПР102) есть авария одного из датчиков.*)
	osmosManager: RichTwoPumpManager;
	toNextStartOsmos1timer: WORD;
	toNextStartOsmos2timer: WORD;
	minutesOfWorkOsmos2: WORD;
	secondsOfWorkOsmos2: WORD;
	osmos1SensorAlarm: BOOL;		(*Авария оборудования основного осмоса.*)
	osmos1EquipmentAlarm: BOOL;		(*Авария оборудования основного осмоса.*)
	osmos2EquipmentAlarm: BOOL;		(*авария оборудования резервного осмоса*)
	tofValve12: TOF;
	tonValve14: TON;
	tofValve14: TOF;
	tonValve18: TON;
	startP0302: BOOL;		(*сигнал на запуск насосов-дозаторов Р03.02*)
	tonPT030101: TON;
	lowPT030101_P030101: BOOL;		(*давление на РТ030101 не достигло значения для старта при
			активном насосе Р03.01/01*)
	lowPT030101_P030102: BOOL;		(*давление на РТ030101 не достигло значения для старта при
			активном насосе Р03.01/02*)
	tonSwitchValve1413: TON;
	valve1413switcher: IfBOOL;
	delayToSwitchValve14to13: TOF;
	F_P030601: PID;		(*PID регулятор по расходу Р03.06/01*)
	P_P030601: PID;		(*PID регулятор по давлению Р03.06/01*)
	Yout_F_P030601: REAL;		(*задание ПИД по расходу для Р030601*)
	Yout_P_P030601: REAL;		(*выход регулировки по давлению Р03.06/01, 0...100*)
	Yout_Total_P030601: REAL;		(*итоговый управляющий сигнал производительность Р03.06/01*)
	Yout_F_P030602: REAL;		(*задание ПИД по расходу для Р030602*)
	Yout_P_P030602: REAL;		(*выход регулировки по давлению Р03.06/02, 0...100*)
	Yout_Total_P030602: REAL;		(*итоговый управляющий сигнал производительность Р03.06/02*)
	P030601alarm: BOOL;		(*авария насоса Р03.06/01*)
	P030602alarm: BOOL;		(*авария насоса Р03.06/02*)
	P030601start: BOOL;		(*сигнал на запуск насоса Р03.06/01*)
	P030602start: BOOL;		(*сигнал на запуск насоса Р03.06/02*)
	osmos1AlarmPT030301: BOOL;		(*авария основного осмоса по макс давлению датчика РТ03.03/01*)
	osmos1AlarmPT030401: BOOL;		(*авария основного осмоса по макс давлению датчика РТ03.04/01*)
	osmos2AlarmPT030302: BOOL;		(*авария основного осмоса по макс давлению датчика РТ03.03/02*)
	osmos2AlarmPT030402: BOOL;		(*авария основного осмоса по макс давлению датчика РТ03.04/02*)
	tofValve18: TOF;
	HoldingToEndProcValve: TOF;
	tonValve17: TON;
	tonValve18rez: TON;
	tofValve18rez: TOF;
	tofValve17: TOF;
	tofValve15: TOF;
	lowPT030102_P030101: BOOL;		(*авария насоса Р03.01/01 по низкому давлению РТ03.01/02*)
	lowPT030102_P030102: BOOL;		(*авария насоса Р03.01/02 по низкому давлению РТ03.01/02*)
	PT030102realValue: REAL;		(*давление РТ03.01/02 из DD2*)
	tonSwitchValve1716: TON;
	HoldingToEndProcValveRez: TOF;
	tonPT030102: TON;
	valve1716switcher: IfBOOL;
	delayToSwitchValve17to16: TOF;
	PT030202realValue: REAL;
	PT030302realValue: REAL;
	PT030402realValue: REAL;
	FIT030302realValue: REAL;
	F_P030602: PID;
	P_P030602: PID;
	FIT030202realValue: REAL;
	QIT030102realValue: REAL;
	freqP030601: LIN_TRAFO;
	freqP030602: LIN_TRAFO;
	pt030102:ControlAI;
	pt030202: ControlAI;
	pt030302: ControlAI;
	pt030402: ControlAI;
	fit0301: ControlAI;
	fit030202: ControlAI;
	qit030102: ControlAI;
	fit030302:ControlAI;
	PT030102alarm: BOOL;		(*авария датчика*)
	PT030202alarm: BOOL;
	PT030302alarm: BOOL;
	PT030402alarm: BOOL;
	FIT0301alarm: BOOL;
	FIT030202alarm: BOOL;
	FIT030302alarm: BOOL;
	QIT030102alarm: BOOL;
	toNextStartP030201timer: WORD;
	toNextStartP030202timer: WORD;
	PT0303setValue: REAL;		(*Задание максимального давления на РТ03.03*)

	testBOOL: BOOL;
	testUINT: UINT;
	testTime: TIME;
	testUIN: UDINT;

	BMTflowToCascade: REAL;		(*Расход в БМТ, от которого рассчитываются уставки расхода
			осмосов 1 и 2, каскадно.*)
	isCascade: BOOL;		(*0 = уставка расходу своя, не каскад
			1 = уставка каскадная от расхода БМТ*)
	OPAN_realStub: WORD;
	OPANboolStub: BOOL;
	OPANsetWordP0301: WORD;		(*****************удалить когда пропишешь переменные удаленной панели*********************************)
	OPANwriteSetWord: WORD;		(************************************************удали когда пропишешь переменные удаленной панели*************************************)
	OPANsetWordP0302: WORD;		(***************************удали после того как пропишешь переменные удаленной панели********************************************)
	OPANsetWordOsmos: WORD;		(********************************удали когда пропишешь переменные удаленной панели********************************)

	onStartCatcher: R_TRIG;

	tof1: TOF;
	tof2: TOF;
	tof3: TOF;
	tof4: TOF;
	tof5: TOF;
	tof6: TOF;
	setWordP0302: WORD;		(*Конфигурация работы доз.насосов Р03.01*)
	setWordOsmos: WORD;		(*Конфигурация режимов работы осмосов*)
	cascadeTrig: RS;
	setCascadeOnStart: IfBOOL;
	highLevelV0207: BOOL;		(*высокий уровень в емкости V02.07*)
	controlAILT0203: ControlAI;
	LT0301alarm: BOOL;		(*авария датчика  LT03.01 уровень в емкости V02.07*)
	LT0302realValue: REAL;		(*уровень в емкости V02.07, м. от датчика LT02.03*)

END_VAR
VAR RETAIN
	counterP030201: DWORD;
	counterP030202: DWORD;
	daysOfWorkP030201: WORD;
	daysOfWorkP030202: WORD;
	hoursOfWorkP030201: WORD;
	hoursOfWorkP030202: WORD;
	minutesOfWorkP030201: WORD;
	minutesOfWorkP030202: WORD;
	secondsOfWorkP030202: WORD;

	counterOsmos1: DWORD;
	counterOsmos2: DWORD;
	daysOfWorkOsmos1: WORD;
	hoursOfWorkOsmos1: WORD;
	minutesOfWorkOsmos1: WORD;
	secondsOfWorkOsmos1: WORD;
	daysOfWorkOsmos2: WORD;
	hoursOfWorkOsmos2: WORD;
	secondsOfWorkP030201: WORD;
	statWordP0301: WORD;		(*статусы состояния насосов Р03.01*)
	statWordP0302: WORD;		(*Статусы состояния доз.насосов Р03.02 на входе осмос 2.*)
	statWordOsmos: WORD;		(*статус состояни осмосов*)
	setWordP0301onStart: WORD;
	setWordP0302onStart: WORD;
	setWordOsmosOnStart: WORD;
	isCascadeOnStart: BOOL;
	FIT0303_SetCascade: REAL;
	PT0301startValue: REAL;		(*Давление РТ0301 для запуска насоса*)
	FIT0303setValue: REAL;		(*Задание расхода для осмоса*)
	PT0302setMaxValue: REAL;
	PT0303setMaxValue: REAL;		(*Задание максимального давления на РТ03.03*)
	PT0304setMaxValue: REAL;
	KP_F_P030601: REAL := 1;
	I_F_P030601: REAL := 10;
	D_F_P030601: REAL := 1;
	KP_P_P030601: REAL := 1;
	I_P_P030601: REAL := 10;
	D_P_P030601: REAL := 1;
	KP_F_P030602: REAL := 1;
	I_F_P030602: REAL := 10;
	D_F_P030602: REAL := 1;
	KP_P_P030602: REAL := 1;
	I_P_P030602: REAL := 10;
	D_P_P030602: REAL := 1;
	setMaxPumpDosingValueP0302: REAL;		(*задание максимальной производительности доз.насоса, в мл/мин*)
	setKoeffProportionalityP0302: REAL;		(*Задание мл на кубометр (коэф.пропорциональности между расходом и дозированием)*)
	CHECKING_DELAY_TIME: TIME;		(*время задержки начала контроля параметра (например, задержка
			контроля эк.манометра после насоса, время на разгон).*)
	DELAY_REPEATED_START_SEC: WORD;		(*время задержки повторного пуска насосов, сек, защита от частых пусков*)
	DELAY_TO_OFF_VALVE: TIME;
	DELAY_TO_CHECK_PT0301: TIME;
	DELAY_TO_SWITCH_VALVE: TIME;		(*время задержки до переключения клапанов после запуска насоса Р0306*)
	DELAY_TO_CLOSE_VALVE: TIME;		(*задержка до начала закрытия клапанов после выключения насосов*)
	FIT0301maxValue: REAL;
	FIT030201maxValue: REAL;
	FIT030301maxValue: REAL;
	FIT030202maxValue: REAL;
	FIT030302maxValue: REAL;
	QIT030101maxValue: REAL;
	QIT030102maxValue: REAL;
	PT030101maxValue: REAL;		(*Максимальное значение показаний датчика РТ03.01/01
			(при 20мА)*)
	PT030201maxValue: REAL;
	PT030301maxValue: REAL;
	PT030401maxValue: REAL;
	PT030102maxValue: REAL;
	PT030202maxValue: REAL;
	PT030302maxValue: REAL;
	PT030402maxValue: REAL;
	LT0203maxValue: REAL;
	V0207maxHeight: REAL;
	V0207minHeight: REAL;
END_VAR
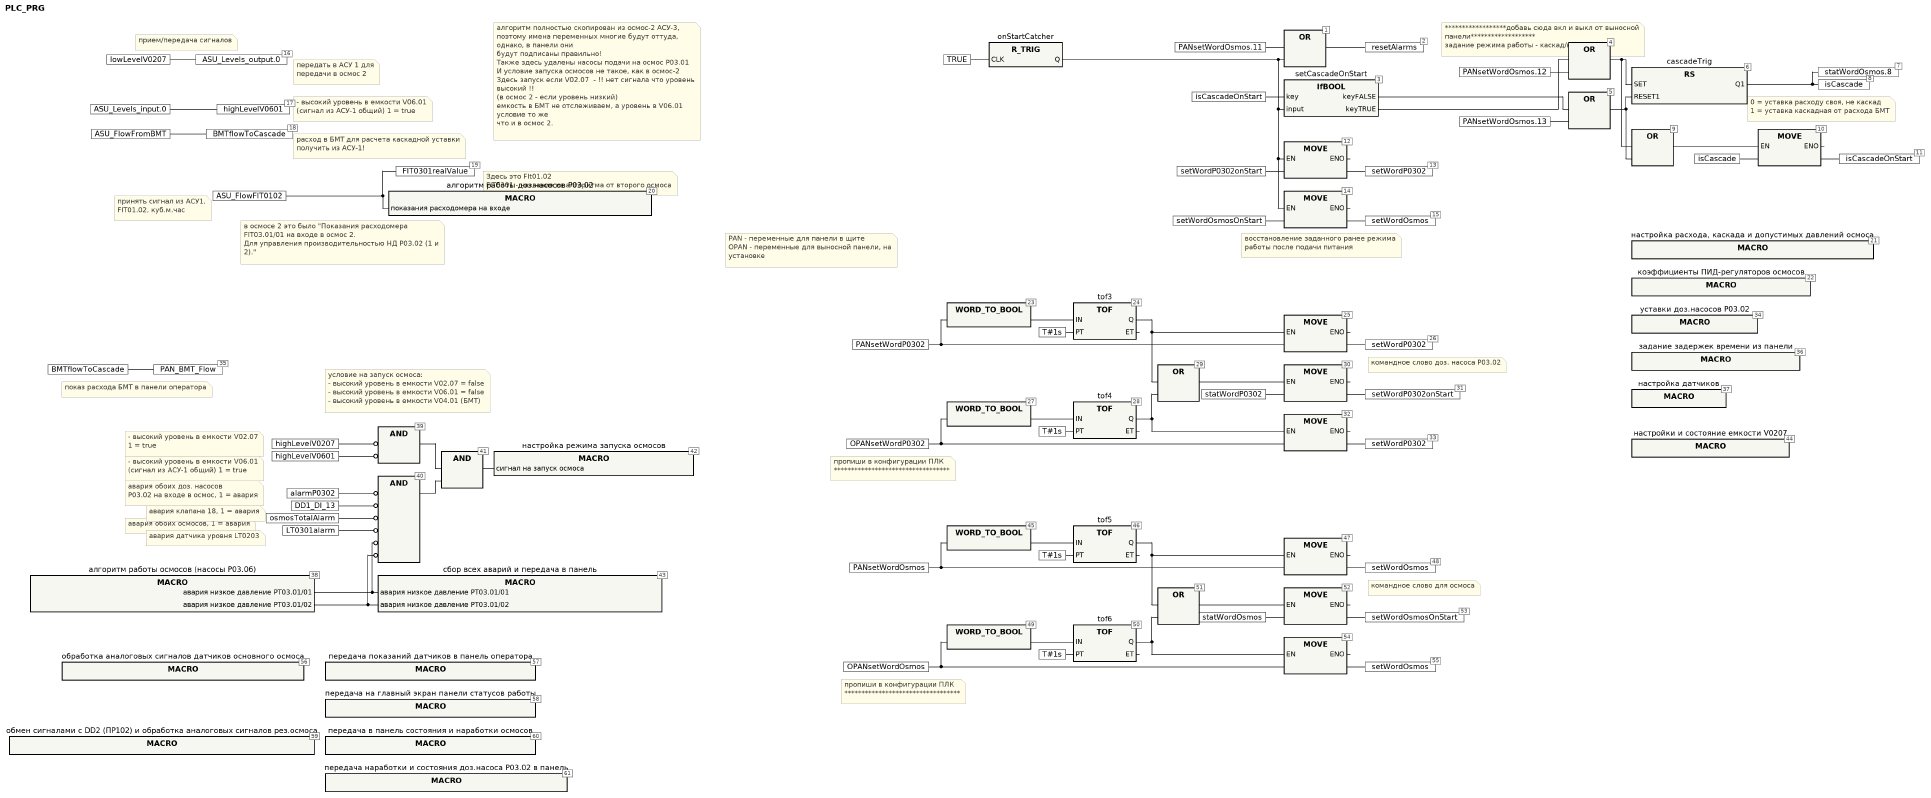
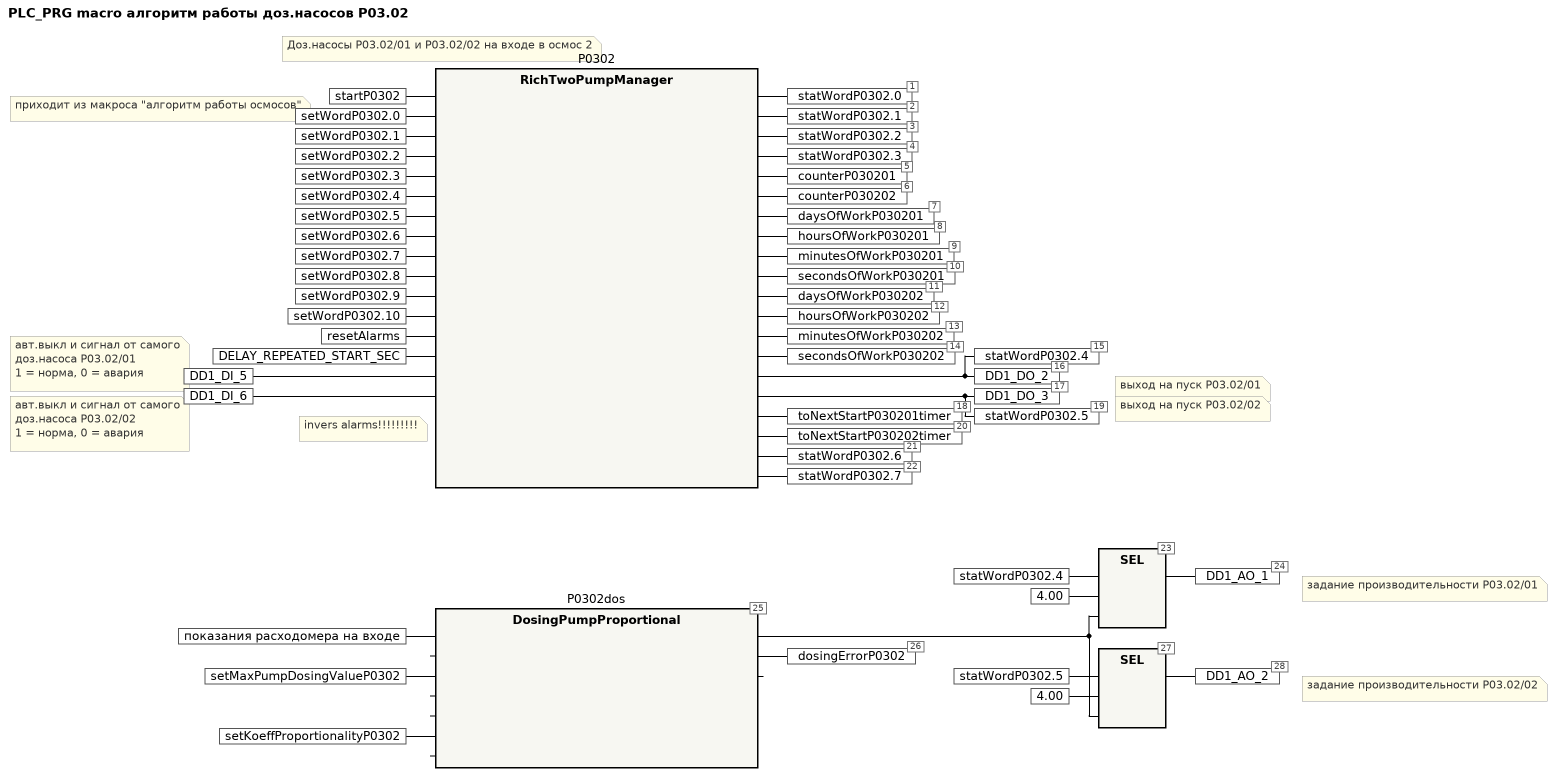
[picture p1: PLC_PRG macro алгоритм работы доз.насосов Р03.02 (CFC)]
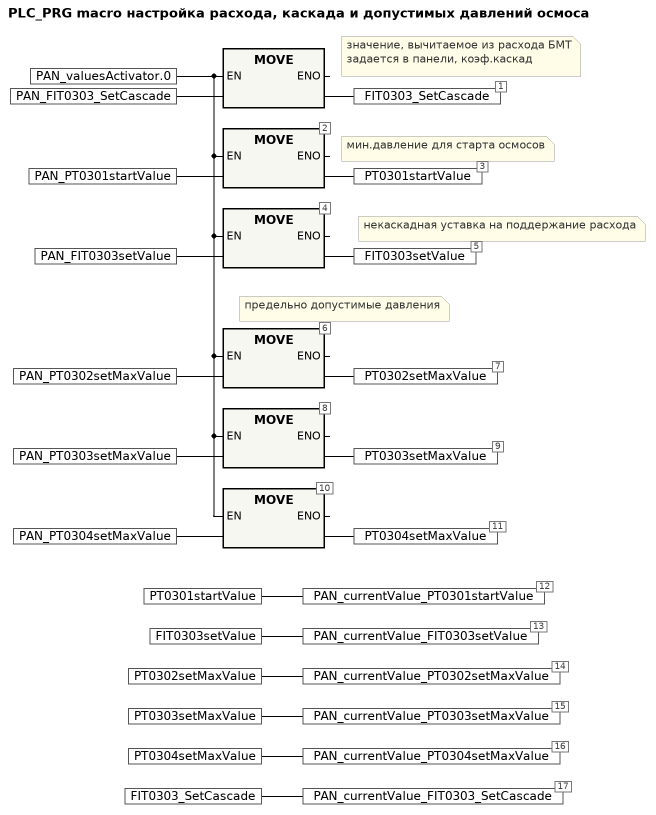
[picture p2: PLC_PRG macro настройка расхода, каскада и допустимых давлений осмоса (CFC)]
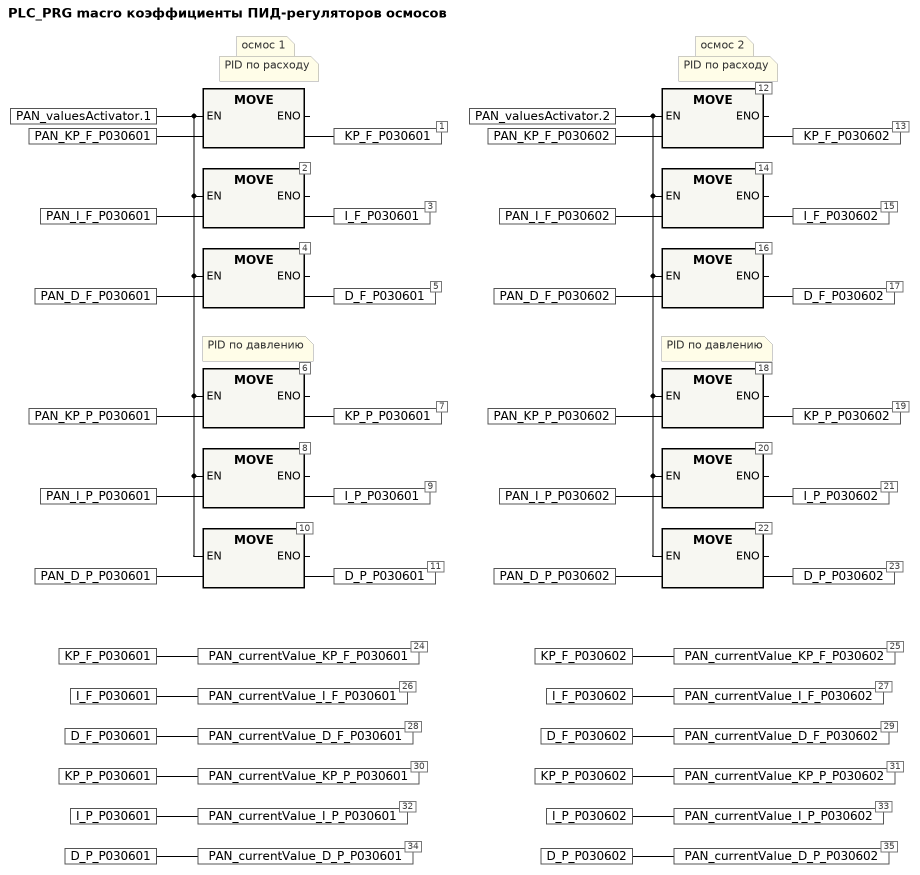
[picture p3: PLC_PRG macro коэффициенты ПИД-регуляторов осмосов (CFC)]
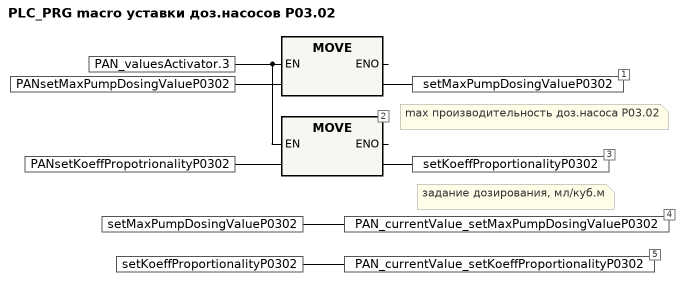
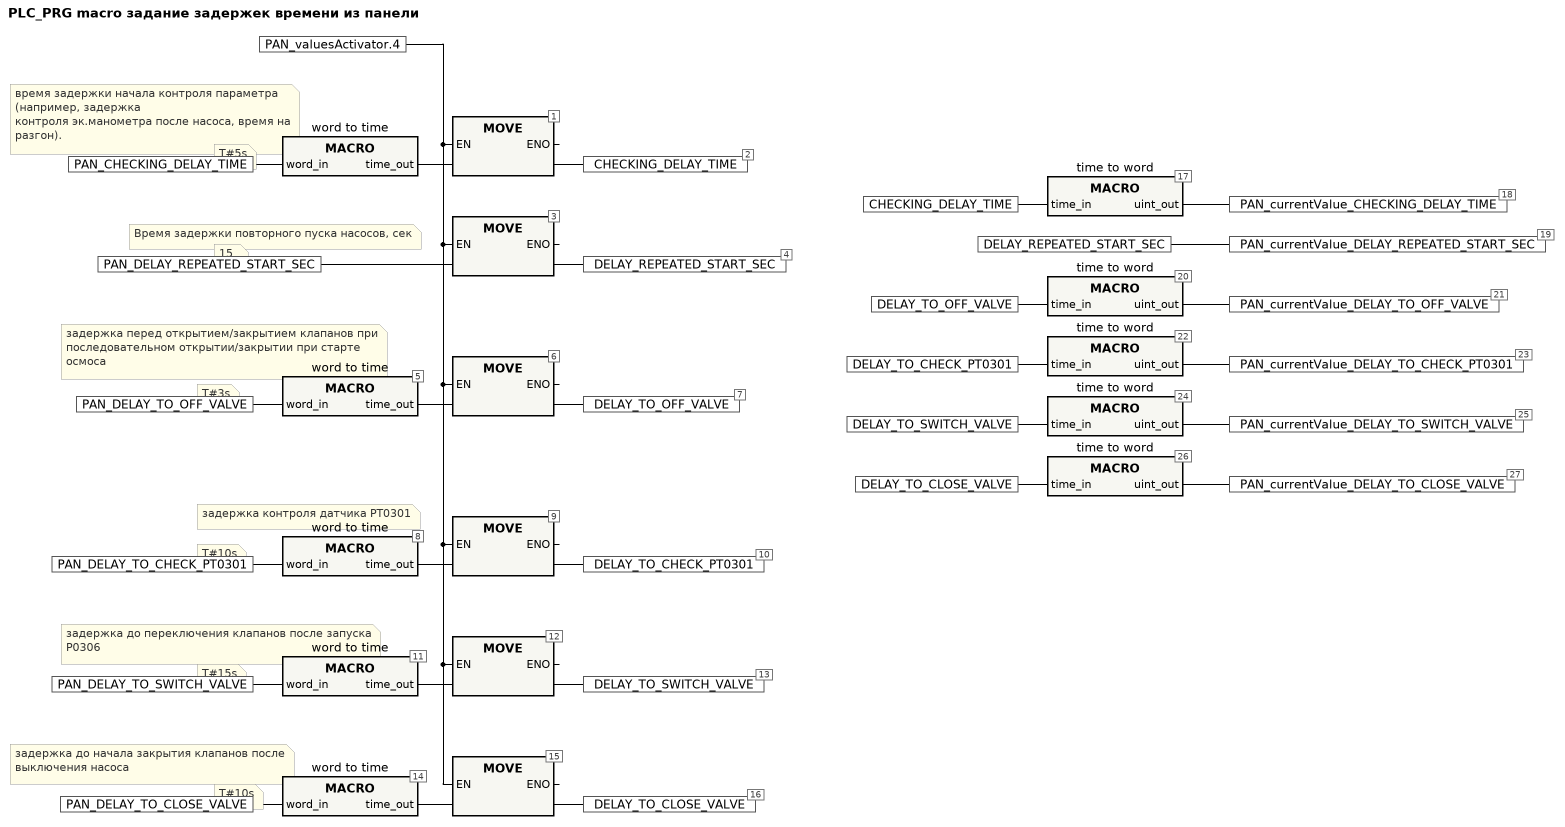
[picture p5: PLC_PRG macro задание задержек времени из панели (CFC)]
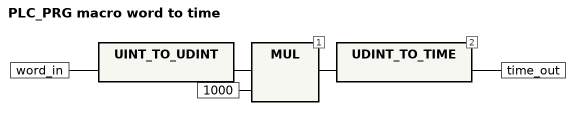
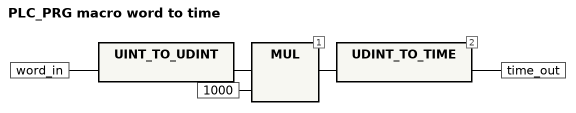
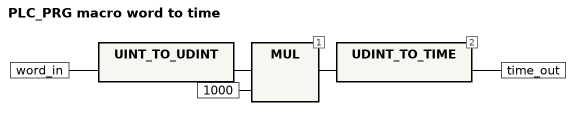
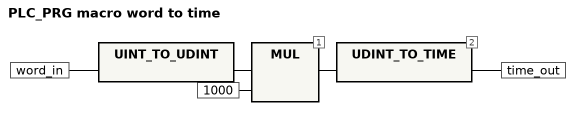
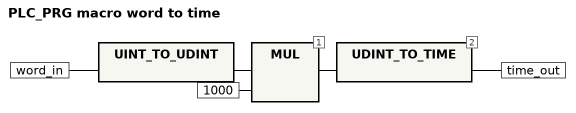
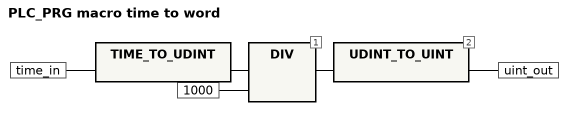
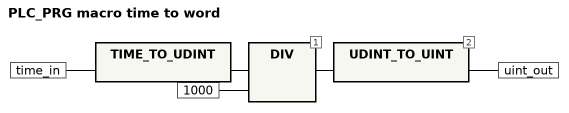
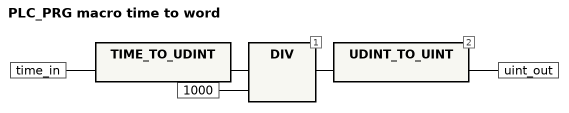
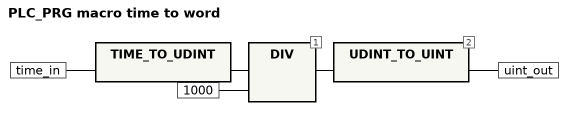
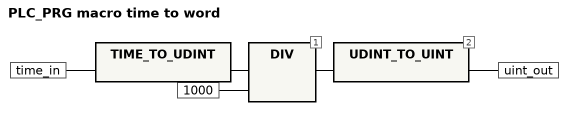
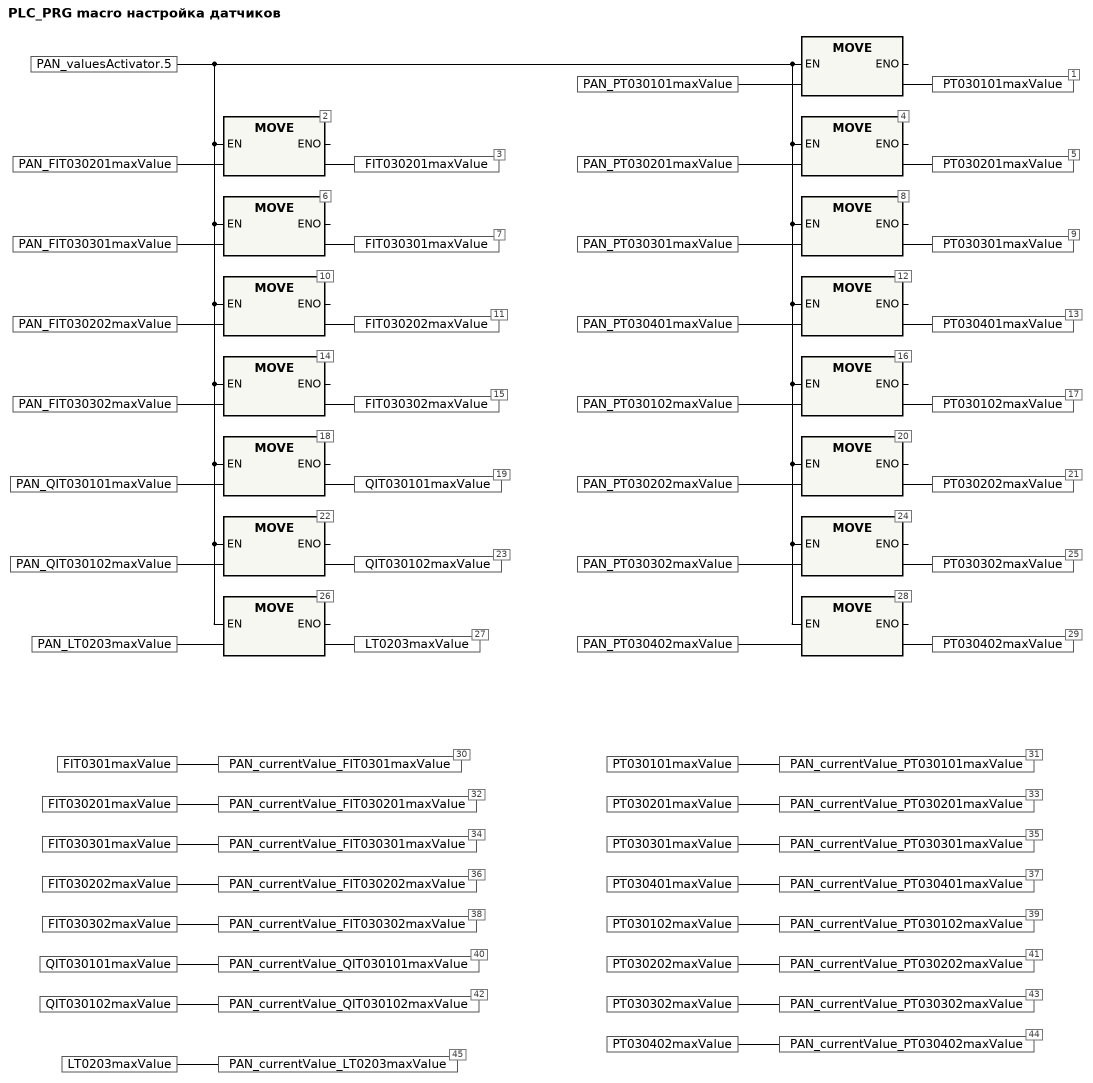
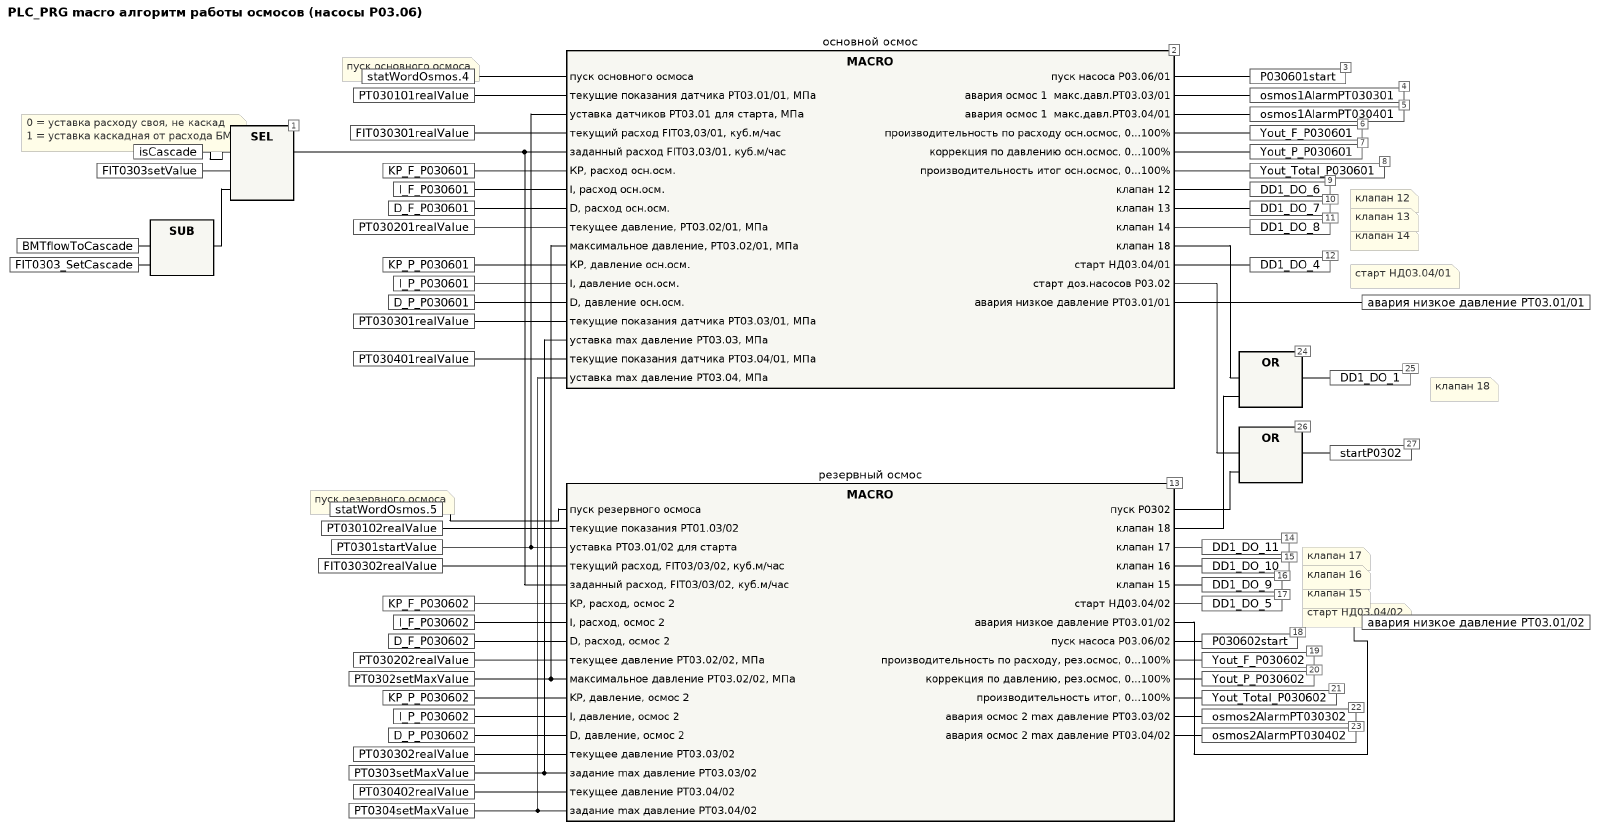
[picture p17: PLC_PRG macro алгоритм работы осмосов (насосы Р03.06) (CFC)]
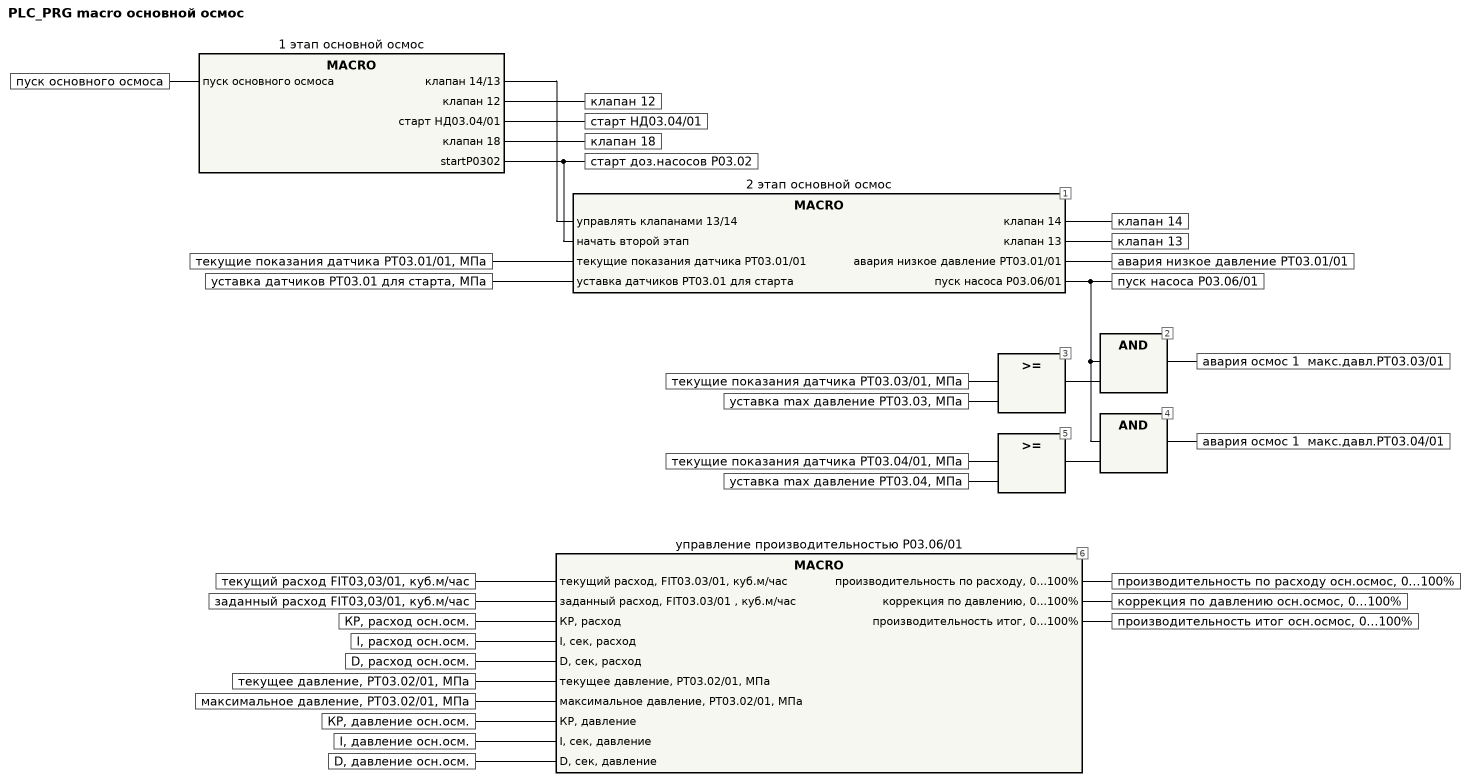
[picture p18: PLC_PRG macro основной осмос (CFC)]
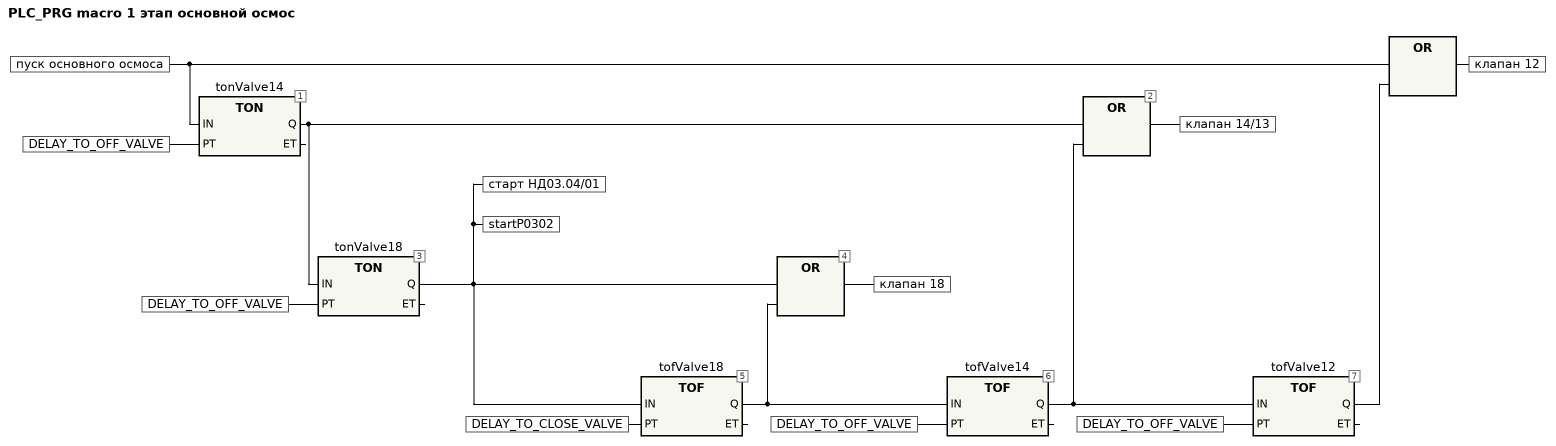
[picture p19: PLC_PRG macro 1 этап основной осмос (CFC)]
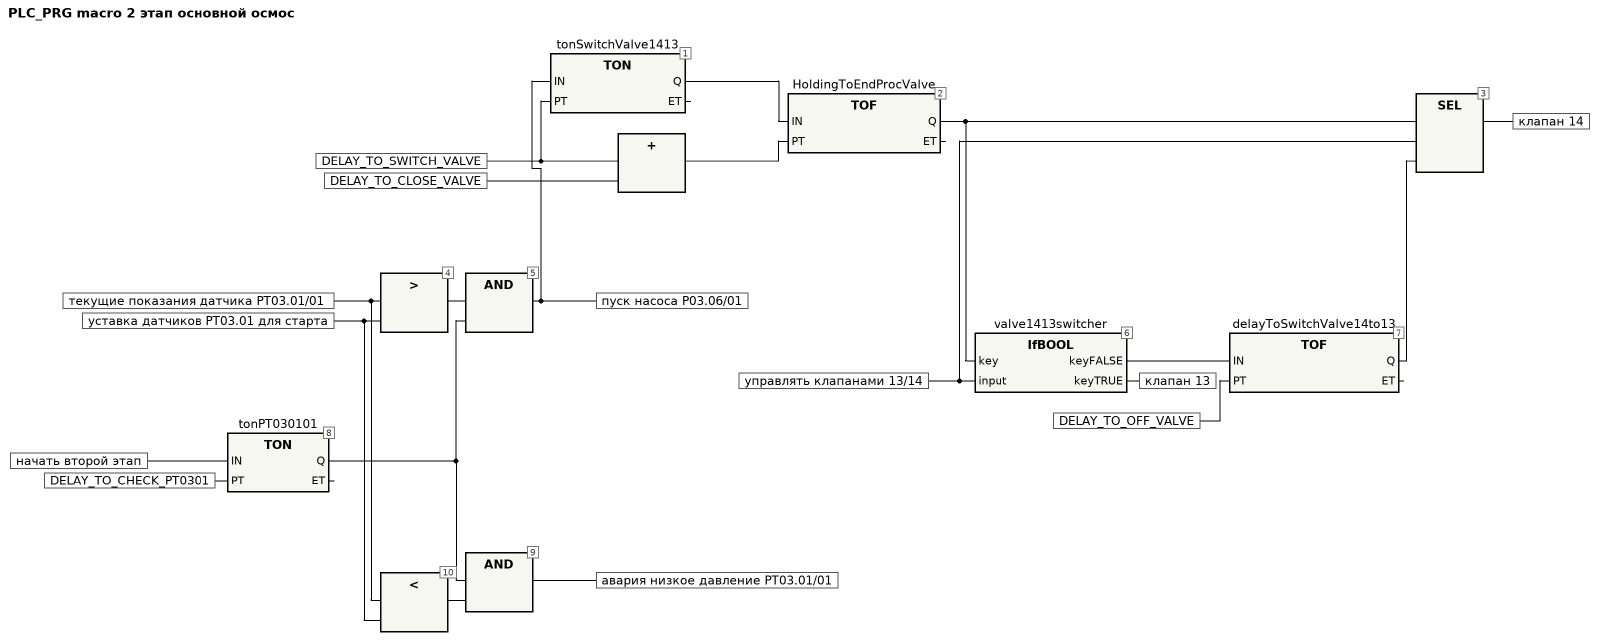
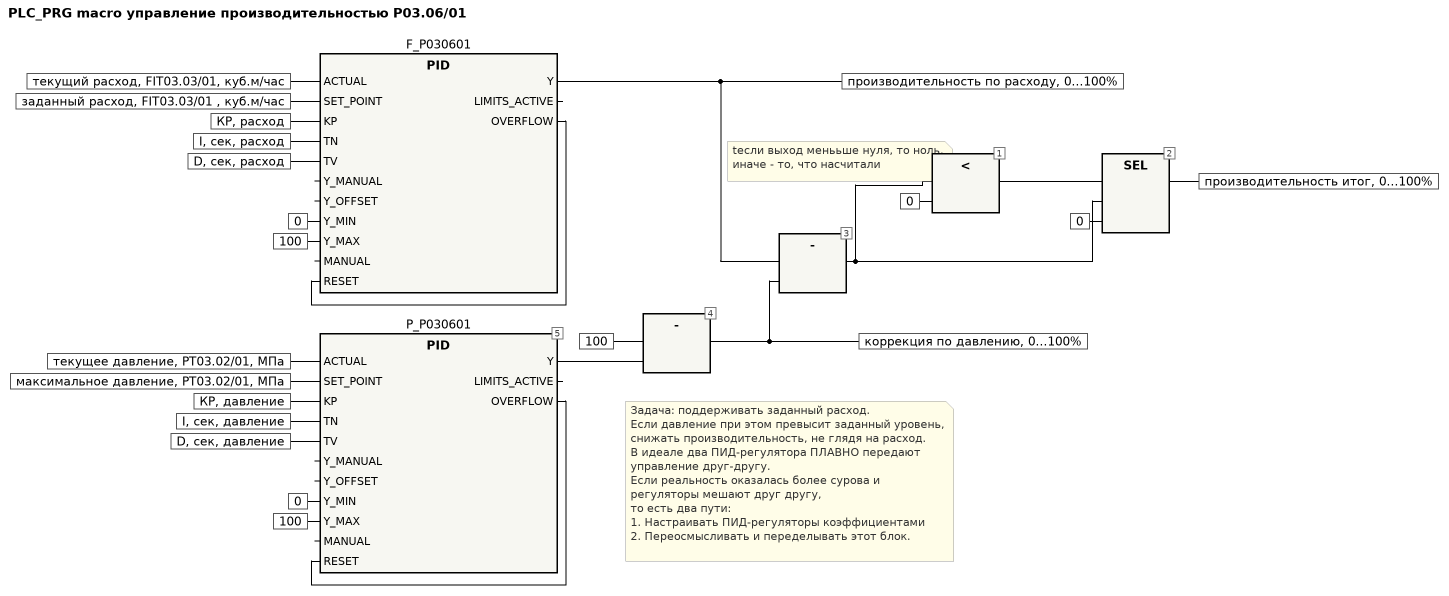
[picture p21: PLC_PRG macro управление производительностью Р03.06/01 (CFC)]
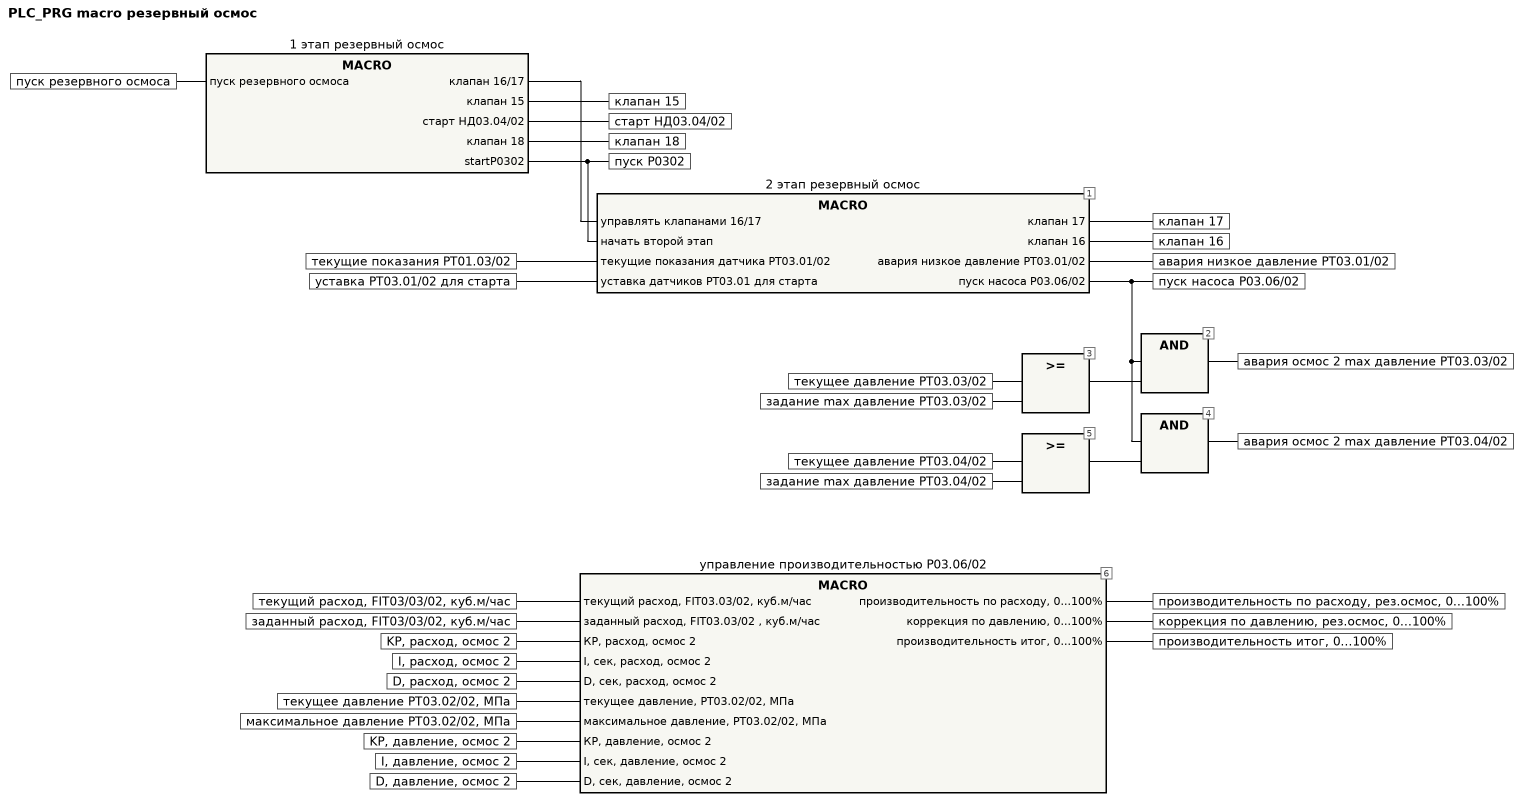
[picture p22: PLC_PRG macro резервный осмос (CFC)]
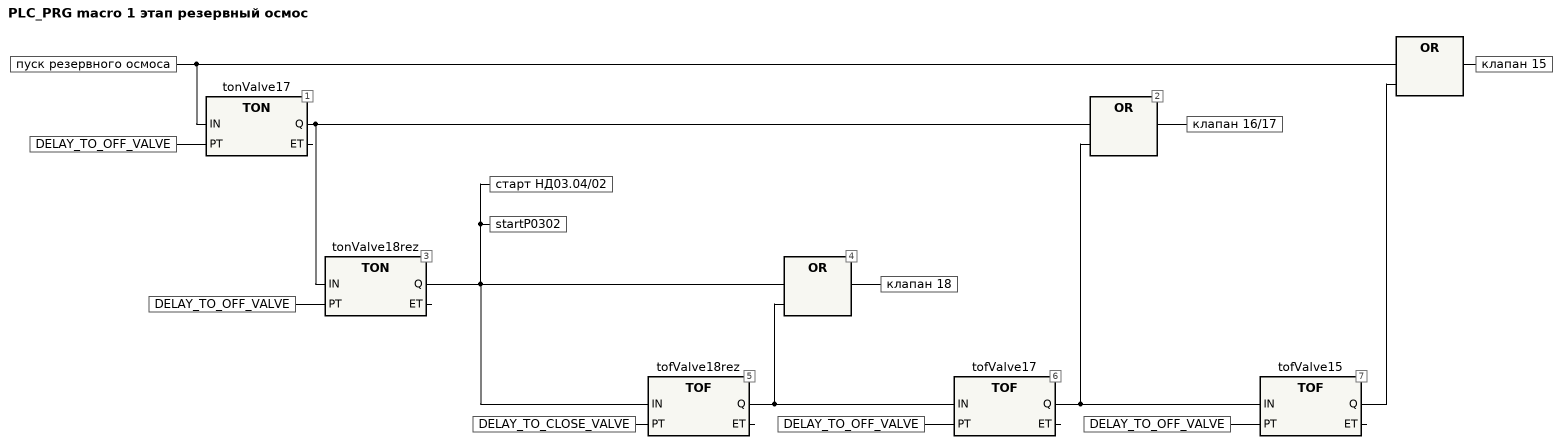
